PROGRAM Axis02_Auto
VAR
//System_Bit
	Always_ON	:	BOOL	:=TRUE	;//상시 ON 
	Always_OFF	:	BOOL	:=FALSE	;//상시 OFF
END_VAR

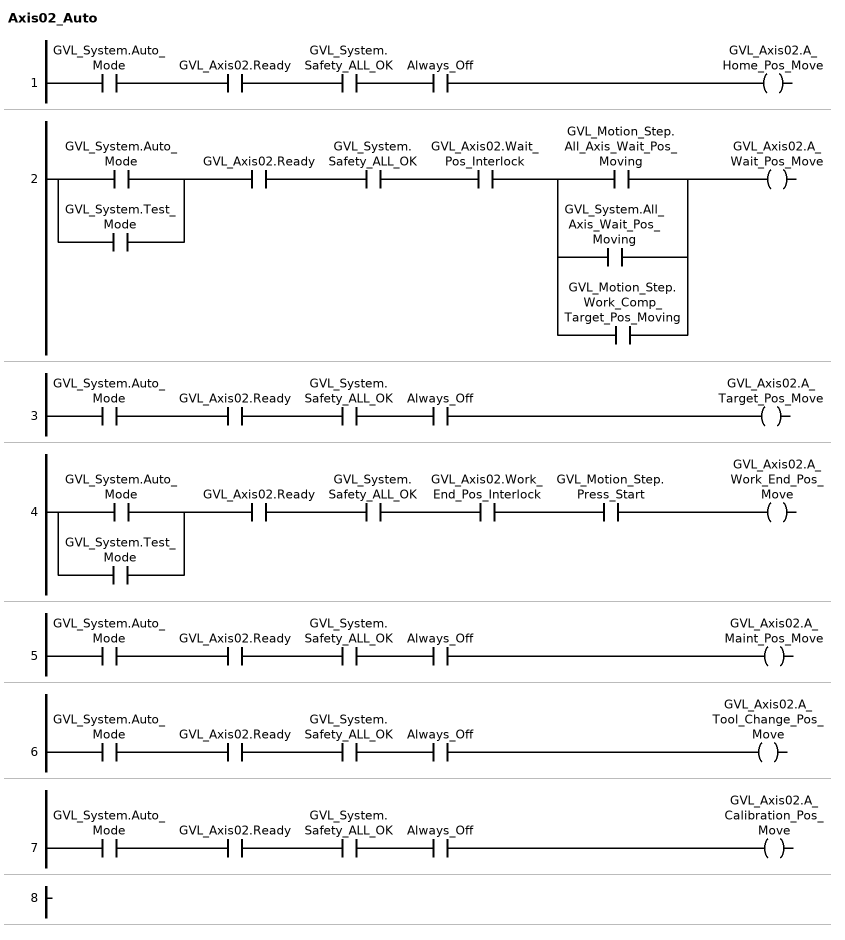
// NETWORK 1
GVL_Axis02.A_Home_Pos_Move := GVL_System.Auto_Mode AND GVL_Axis02.Ready AND GVL_System.Safety_ALL_OK AND Always_Off;

// NETWORK 2
GVL_Axis02.A_Wait_Pos_Move := (GVL_System.Auto_Mode OR GVL_System.Test_Mode) AND GVL_Axis02.Ready AND GVL_System.Safety_ALL_OK AND GVL_Axis02.Wait_Pos_Interlock AND (GVL_Motion_Step.All_Axis_Wait_Pos_Moving OR GVL_System.All_Axis_Wait_Pos_Moving OR GVL_Motion_Step.Work_Comp_Target_Pos_Moving);

// NETWORK 3
GVL_Axis02.A_Target_Pos_Move := GVL_System.Auto_Mode AND GVL_Axis02.Ready AND GVL_System.Safety_ALL_OK AND Always_Off;

// NETWORK 4
GVL_Axis02.A_Work_End_Pos_Move := (GVL_System.Auto_Mode OR GVL_System.Test_Mode) AND GVL_Axis02.Ready AND GVL_System.Safety_ALL_OK AND GVL_Axis02.Work_End_Pos_Interlock AND GVL_Motion_Step.Press_Start;

// NETWORK 5
GVL_Axis02.A_Maint_Pos_Move := GVL_System.Auto_Mode AND GVL_Axis02.Ready AND GVL_System.Safety_ALL_OK AND Always_Off;

// NETWORK 6
GVL_Axis02.A_Tool_Change_Pos_Move := GVL_System.Auto_Mode AND GVL_Axis02.Ready AND GVL_System.Safety_ALL_OK AND Always_Off;

// NETWORK 7
GVL_Axis02.A_Calibration_Pos_Move := GVL_System.Auto_Mode AND GVL_Axis02.Ready AND GVL_System.Safety_ALL_OK AND Always_Off;

// NETWORK 8

END_PROGRAM

(* stored: Version 1.1.0.1, ProductVersion 3.1.4024.15
   POU Axis02_Auto: Id {bb8b8c2e-2fd8-4db4-a00c-53cc54166e35}, SpecialFunc None *)
